(* CoDeSys 2.3.9.47 project: myFirstPID.pro *)
(* Libraries: STANDARD.LIB 5.6.98 11:03:02 *)

(* Task configuration *)
TASK Standard (PRIORITY := 0, INTERVAL := T#10ms);
	MAIN
END_TASK

(* Global variable list: Global_Variables *)
VAR_GLOBAL
t_cycle : REAL;
t_global: REAL;
T_sample: REAL;
END_VAR

(* Data type *)
TYPE PID_parameters :
STRUCT
(*Essential Parameters*)
Kp			:REAL;
Ti			:REAL;
Td			:REAL;
N			:REAL;
sat_high	:REAL;
sat_low		:REAL;

(*Features*)
has_arw	:BOOL;
has_sat	:BOOL;
has_bra	:BOOL;

END_STRUCT
END_TYPE

(* Data type *)
TYPE PT1T2_parameters :
STRUCT
K	: REAL;
T_1	: REAL;
T_2	: REAL;
END_STRUCT
END_TYPE

(* Data type *)
TYPE System_Mode :
(
	STATE_SM_INIT := 0,
	STATE_SM_RUN  := 1
);
END_TYPE

(* POU MAIN, ST *)
PROGRAM MAIN
VAR
(*PID STUFF*)
pid		: PID_Controller;
pid_par	: PID_parameters;
ref		: REAL:= 0;
(*SYSTEM STUFF*)
system	: PT1T2;
mode	: System_Mode := STATE_SM_INIT;
sys_par	: PT1T2_parameters;
END_VAR
t_cycle := 0.01;
T_sample := t_cycle;



CASE mode OF
	STATE_SM_INIT :
(*
*)
(*System Parameters*)
sys_par.K 	:= 10;
sys_par.T_1	:= 0.1;
sys_par.T_2	:= 0.01;

(*Initialize System*)
system();
system.mode := mode;

(*Essential PID Parameters*)
pid_par.Kp			:=  1/sys_par.K;
pid_par.Ti			:=  sys_par.T_1;
pid_par.Td			:=  sys_par.T_2;
pid_par.N			:=  100;
pid_par.sat_high	:=  100;
pid_par.sat_low		:= -100;
(*PID Features*)
pid_par.has_arw	:= FALSE;
pid_par.has_sat	:= FALSE;
pid_par.has_bra	:=  TRUE;

(*Initialize Controller*)
pid();
pid.param := pid_par;
(*Actualize Mode*)
mode := STATE_SM_RUN;
(*
*)
	STATE_SM_RUN  :
(*
*)
system.mode := mode;
pid.r_k := ref;
system.x_k := pid.u_k;
pid.y_k := system.y_k;
pid();
system();
(*
*)
ELSE
	mode := STATE_SM_INIT;
END_CASE;


(*Increment global Time*)
t_global := t_global + t_cycle;
END_PROGRAM

(* POU PID_Controller, ST *)
FUNCTION_BLOCK PID_Controller
VAR_INPUT
	r_k		: REAL;
	y_k		: REAL;
	param	: PID_parameters;
END_VAR
VAR_OUTPUT
	u_k		: REAL;
END_VAR
VAR
	e_k		: REAL:= 0;
	e_k_1	: REAL;
	(*P-Part*)
	u_p_k	: REAL:= 0;
	(*I-Part*)
	u_i_k	: REAL:= 0;
	u_i_k_1	: REAL;
	(*D-Part*)
	u_d_k	: REAL:= 0;
	u_d_k_1	: REAL;
	a		: REAL;
	b		: REAL;
END_VAR
(*Calculate Error*)
e_k := r_k - y_k;
e_k := e_k * param.Kp;

a 	:= param.Td / (param.Td + param.N * t_cycle);
b	:= (param.Kp * param.Td * param.N)/(param.Td + param.N * t_cycle);

(*Proportional Term*)
u_p_k := e_k;

(*Integrator using Trapeze Approximation*)
u_i_k := u_i_k_1 + (e_k + e_k_1)*t_cycle/(2*param.Ti);

(*Derivate Term*)
IF (param.has_bra = TRUE) THEN
u_d_k := param.Kp * param.Td * (-y_k - e_k_1) / t_cycle;
ELSE
u_d_k := -(a*u_d_k_1 + b*(e_k - e_k_1));
END_IF

(*Calculate Output*)
PID_Controller.u_k := u_p_k + u_i_k + u_d_k;

(*Actualize later used Variables*)
e_k_1 	:= e_k;
u_i_k_1 := u_i_k;
u_d_k_1	:= u_d_k;
END_FUNCTION_BLOCK

(* POU PT1T2, ST *)
FUNCTION_BLOCK PT1T2
VAR_INPUT
x_k		: REAL;
param	: PT1T2_parameters;
mode	: System_Mode;
END_VAR
VAR_OUTPUT
y_k		: REAL;
END_VAR
VAR
x_k_1	: REAL;
x_k_2	: REAL;
y_k_1	: REAL;
y_k_2	: REAL;
(*Coefficients*)
a1		: REAL;
a2		: REAL;
b0		: REAL;
b1		: REAL;
c1		: REAL;
c2		: REAL;
END_VAR
CASE mode OF
	STATE_SM_INIT :
		(*Calculation of Coefficients*)
		a1 := EXP(-T_sample/param.T_1);
		a2 := EXP(-T_sample/param.T_2);
		b0 := (param.T_1*(1-a1)-param.T_2*(1-a2))*param.K/(param.T_1 - param.T_2);
		b1 := (param.T_2*a1*(1-a2)-param.T_1*a2*(1-a1))*param.K/(param.T_1 - param.T_2);
		c1 := -(a1+a2);
		c2 := a1*a2;

	STATE_SM_RUN  :
		y_k := b0*x_k_1 + b1*x_k_2 + c1*y_k_1 + c2*y_k_2;
ELSE
	mode := STATE_SM_INIT;
END_CASE;
END_FUNCTION_BLOCK
